// TIA Portal V17 export
// export: Created 2024-08-07T21:43:52.7889456Z, ExportSetting WithDefaults, DisplayName Totally Integrated Automation Portal, DisplayVersion V17 Update 7, DisplayName TIA Portal Openness, DisplayVersion V17 Update 7, DisplayName TIA Portal Version Control Interface, DisplayVersion V17, DisplayName SINAMICS Startdrive Advanced, DisplayVersion V17 SP2, DisplayName SINAMICS Startdrive G110M, G120, G120C, G120D, G120P, G115D, DisplayVersion V17 SP2, DisplayName SINAMICS Startdrive G130, G150, S120, S150, SINAMICS MV, S210, DisplayVersion V17 SP2, DisplayName STEP 7 Professional, DisplayVersion V17 Update 7, DisplayName STEP 7 Safety, DisplayVersion V17 Update 6, DisplayName WinCC Advanced / Unified PC, DisplayVersion V17 Update 7
FUNCTION "FC_UIntToBits" : Void   // FC1021, LAD
{ S7_Optimized_Access := 'FALSE' }
VERSION : 0.1
// stored: AutoNumber false, IsIECCheckEnabled false, SetENOAutomatically false, UDAEnableTagReadback false
   VAR_INPUT
      iValue : UInt;
   END_VAR
   VAR_OUTPUT
      qBit1 : Bool;
      qBit2 : Bool;
      qBit3 : Bool;
      qBit4 : Bool;
      qBit5 : Bool;
      qBit6 : Bool;
      qBit7 : Bool;
      qBit8 : Bool;
      qBit9 : Bool;
      qBit10 : Bool;
      qBit11 : Bool;
      qBit12 : Bool;
      qBit13 : Bool;
      qBit14 : Bool;
      qBit15 : Bool;
      qBit16 : Bool;
   END_VAR
   VAR_TEMP
      value : UInt;
   END_VAR
BEGIN

REGION Network 1: Convert UInt to bits
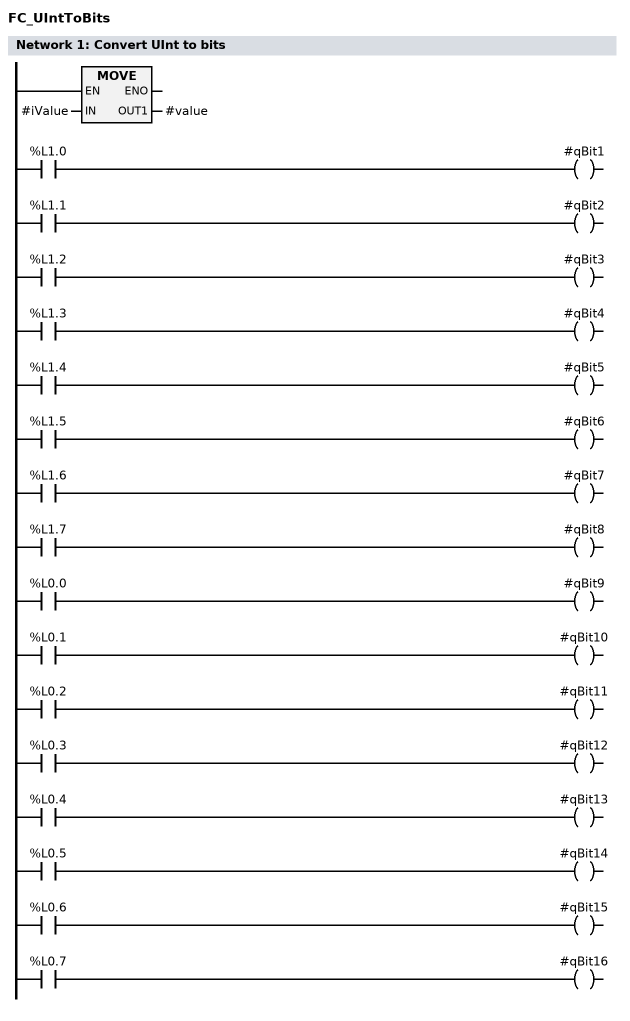
   RUNG wire#powerrail
      Move(in := #iValue, out1 => #value)
   END_RUNG
   RUNG wire#powerrail
      Contact( %L1.0 )
      Coil( #qBit1 )
   END_RUNG
   RUNG wire#powerrail
      Contact( %L1.1 )
      Coil( #qBit2 )
   END_RUNG
   RUNG wire#powerrail
      Contact( %L1.2 )
      Coil( #qBit3 )
   END_RUNG
   RUNG wire#powerrail
      Contact( %L1.3 )
      Coil( #qBit4 )
   END_RUNG
   RUNG wire#powerrail
      Contact( %L1.4 )
      Coil( #qBit5 )
   END_RUNG
   RUNG wire#powerrail
      Contact( %L1.5 )
      Coil( #qBit6 )
   END_RUNG
   RUNG wire#powerrail
      Contact( %L1.6 )
      Coil( #qBit7 )
   END_RUNG
   RUNG wire#powerrail
      Contact( %L1.7 )
      Coil( #qBit8 )
   END_RUNG
   RUNG wire#powerrail
      Contact( %L0.0 )
      Coil( #qBit9 )
   END_RUNG
   RUNG wire#powerrail
      Contact( %L0.1 )
      Coil( #qBit10 )
   END_RUNG
   RUNG wire#powerrail
      Contact( %L0.2 )
      Coil( #qBit11 )
   END_RUNG
   RUNG wire#powerrail
      Contact( %L0.3 )
      Coil( #qBit12 )
   END_RUNG
   RUNG wire#powerrail
      Contact( %L0.4 )
      Coil( #qBit13 )
   END_RUNG
   RUNG wire#powerrail
      Contact( %L0.5 )
      Coil( #qBit14 )
   END_RUNG
   RUNG wire#powerrail
      Contact( %L0.6 )
      Coil( #qBit15 )
   END_RUNG
   RUNG wire#powerrail
      Contact( %L0.7 )
      Coil( #qBit16 )
   END_RUNG
   // the same network as SCL:
   #value := #iValue;
   #qBit1 := %L1.0;
   #qBit2 := %L1.1;
   #qBit3 := %L1.2;
   #qBit4 := %L1.3;
   #qBit5 := %L1.4;
   #qBit6 := %L1.5;
   #qBit7 := %L1.6;
   #qBit8 := %L1.7;
   #qBit9 := %L0.0;
   #qBit10 := %L0.1;
   #qBit11 := %L0.2;
   #qBit12 := %L0.3;
   #qBit13 := %L0.4;
   #qBit14 := %L0.5;
   #qBit15 := %L0.6;
   #qBit16 := %L0.7;
END_REGION
END_FUNCTION
